(* PLC project Senza_nome, Sconosciuto Senza_nome 1 *)
(* stored: creationDateTime 2026-08-25T12:33:32, modificationDateTime 2026-08-25T12:45:44 *)

PROGRAM program0
  VAR
    P1 : BOOL;
    P2 : BOOL;
    K1 : BOOL;
    K2 : BOOL;
    LAMPADA1 : BOOL;
    LAMPADA2 : BOOL;
  END_VAR

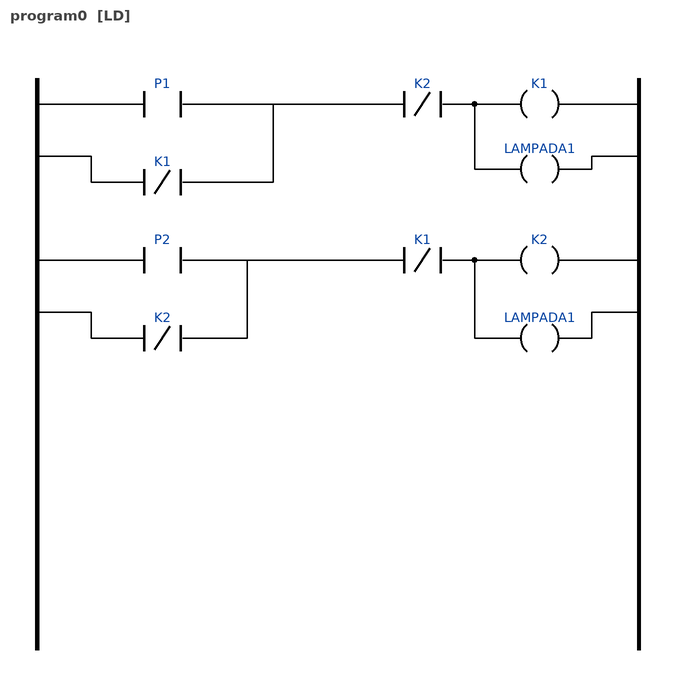
(* LD diagram, written out as Structured Text *)
K1 := (P1 OR NOT K1) AND NOT K2;
K2 := (P2 OR NOT K2) AND NOT K1;
LAMPADA1 := (P1 OR NOT K1) AND NOT K2;
LAMPADA1 := (P2 OR NOT K2) AND NOT K1;
END_PROGRAM

CONFIGURATION Config0
  RESOURCE Res0 ON PLC
    TASK task0(INTERVAL := T#20ms, PRIORITY := 0);
    PROGRAM instance0 WITH task0 : program0;
  END_RESOURCE
END_CONFIGURATION
